FUNCTION_BLOCK FB_OP_MODE_HMI
VAR
	itfOpMode:  I_OP_MODE;
	
//Press 
	bClick_Reset					: BOOL;
	bClick_Start					: BOOL;
	bClick_Stop						: BOOL;
	bClickPause						: BOOL;
	

//State
	bStateStart						: BOOL;
	bStateStop						: BOOL;
	bStatePause						: BOOL;
	bStateReset						: BOOL;
	

//Enable
	bEnableStart					: BOOL:=TRUE;
	bEnableStop						: BOOL:=TRUE;
	bEnablePause					: BOOL:=TRUE;
	bEnableReset					: BOOL:=TRUE;
	
//Options
	bEnableCalibration				: BOOL;
	bOptionCalibration				: BOOL;
	
	bEnableStepByStep				: BOOL;
	bOptionStepByStep				: BOOL;
	
	bEnableEmptyRun					: BOOL;
	bOptionEmptyRun					: BOOL;
	
	
//TextlistID
	nTexlistID						: INT;
	
	fbBlink							: FB_Blink;
END_VAR
VAR_IN_OUT

END_VAR
VAR
END_VAR

IF bClick_Start THEN
	bClick_Start:=FALSE;
	nTexlistID:=nTexlistID+1;
	IF NOT bStateStart THEN
		bStateStart:=TRUE;
		bStateStop:=FALSE;
		bStatePause:=FALSE;
	ELSE
		bStateStart:=FALSE;
	END_IF
END_IF

IF bClick_Stop THEN
	bClick_Stop:=FALSE;
	nTexlistID:=nTexlistID-1;
	IF NOT bStateStop THEN
		bStateStop:=TRUE;
		bStateStart:=FALSE;
		bStatePause:=FALSE;
	ELSE
		bStateStop:=FALSE;
	END_IF
END_IF

IF bClickPause THEN
	bClickPause:=FALSE;
	nTexlistID:=nTexlistID+1;
	IF NOT bStateStop THEN
		bStatePause:=TRUE;
		bStateStop:=FALSE;
		bStateStart:=FALSE;
	ELSE
		bStatePause:=FALSE;
	END_IF
END_IF

METHOD FB_init : BOOL
VAR_INPUT
	bInitRetains : BOOL; // if TRUE, the retain variables are initialized (warm start / cold start)
	bInCopyCode : BOOL;  // if TRUE, the instance afterwards gets moved into the copy code (online change)
	itfOpMode:  I_OP_MODE;
END_VAR
this^.itfOpMode:= itfOpMode;
END_METHOD

END_FUNCTION_BLOCK

(* stored: Version 1.1.0.1, ProductVersion 3.1.4024.12
   POU FB_OP_MODE_HMI: Id {f51e3441-7f47-4cc8-b64b-3e87b9320d78}, SpecialFunc None
   Method FB_init: Id {e2ba2658-016e-42ca-a314-bd82a8b399a2} *)
